Staubli VAL3: sendData.pgx

public program sendData(sio& x_sTcpSocket (dimensions=1), num& x_nData[] (dimensions=1), num& x_nFlag (dimensions=1))
  local num l_nRetVal
begin
  // send data via socket connection...
  // but only if connection is alive, or
  // if heartbeat is not expected
  if (x_nFlag==1 or bCheckHeartbeat==false)
    l_nRetVal=sioSet(x_sTcpSocket,x_nData)
    if (l_nRetVal==-1)
      if (x_nFlag==1)
        x_nFlag=-1
      endIf
    elseIf (l_nRetVal<size(x_nData))
      popUpMsg("Error while sending data")
      x_nFlag=-1
    elseIf (bCheckHeartbeat==false)
      // once data is sent over an open connection,
      // flag it as connected...
      // however, it will never be possible to detect
      // disconnections because the status goes into
      // CLOSE_WAIT, but sioSet() keeps writing data
      // to the socket...
      x_nFlag=1
    endIf
  endIf
end
